TEXTLIST TextList
  0 = 'Manual' | Korea: '수동' | English: 'Manual'
  1 = 'Auto' | Korea: '자동' | English: 'Auto'
   = ''
END_TEXTLIST

(* stored: Version 1.1.0.1
   TextList TextList: Id {efce2b2c-ce8b-489d-89b2-d1bc9b843e07} *)
